Universal Robots PolyScope program: Alinear en base.urp

Program Alinear en base (installation=default directory=/programs/usbdisk createdIn=3.15.1.106171 lastSavedIn=3.15.1.106171 robotSerialNumber=2016353899)
Calibrated DH parameters: a=[0.000013, -0.400736, -0.391774, 0.000067, 0.000127, 0]; d=[0.089273, 42.382267, -41.145698, -1.126577, 0.094921, 0.082461]; alpha=[1.570429, -0.003356, 0.01464, 1.57092, -1.570909, 0]; deltaTheta=[0.000009, -0.341028, 0.387244, -0.046195, -0.000051, -0.000108]
BeforeStart
  Script file /programs/alinearrobot.script
    | def alinearRobot(pose_actual):
    | target_pose=p[0,0,0,0,0,0]
    | rotRPY = [0,0,0]
    | rotRotvec = [0,0,0]
    | rotRPY=rotvec2rpy([pose_actual[3],pose_actual[4],pose_actual[5]])
    | rotRPY[0]=d2r(0)
    | rotRPY[1]=d2r(180)
    | rotRotvec=rpy2rotvec(rotRPY)
    | target_pose[0]=pose_actual[0]
    | target_pose[1]=pose_actual[1]
    | target_pose[2]=pose_actual[2]
    | target_pose[3]=rotRotvec[0]
    | target_pose[4]=rotRotvec[1]
    | target_pose[5]=rotRotvec[2]
    | 
    | return target_pose
    | end
  MoveJ speed 60 deg/s, acceleration 80 deg/s^2 (useActiveTCP=true)
    Waypoint Punto_de_paso_1: TCP in base x=-273.764 y=389.901 z=125.189 mm, rx=1.1525 ry=-1.1848 rz=-0.9862 rad; joints [-78.816, -71.928, 116.512, -57.584, 4.233, 22.466] deg
    SuppressedNode
      rotacionRPY := [0,0,0]
    SuppressedNode
      rotacionRotvec := [0,0,0]
Robot Program (runOnlyOnce=false)
  SuppressedNode
    Folder Carpeta
      pos := get_actual_tcp_pose()
      Script: rotacionRPY=rotvec2rpy([pos[3],pos[4],pos[5]])
      Script: rotacionRPY[0]=d2r(0)
      Script: rotacionRPY[1]=d2r(180)
      Script: rotacionRotvec=rpy2rotvec([rotacionRPY[0],rotacionRPY[1],rotacionRPY[2]])
      Script: pos[3]=rotacionRotvec[0]
      Script: pos[4]=rotacionRotvec[1]
      Script: pos[5]=rotacionRotvec[2]
      target := p[pos[0],pos[1],pos[2],pos[3],pos[4],pos[5]]
  Script: target=alinearRobot(get_actual_tcp_pose())
  MoveJ speed 60 deg/s, acceleration 80 deg/s^2 (useActiveTCP=true)
    Waypoint Punto_de_paso (Variable): variable=target
  Wait Sleep waitTime=2
  MoveJ speed 60 deg/s, acceleration 80 deg/s^2 (useActiveTCP=true)
    Waypoint Punto_de_paso_1: TCP in base x=-273.764 y=389.901 z=125.189 mm, rx=1.1525 ry=-1.1848 rz=-0.9862 rad; joints [-78.816, -71.928, 116.512, -57.584, 4.233, 22.466] deg
